(* Logix 5000 project; controller StackLight_Jimmy vendor 1 type 14 code 158 rev 27.11; software revision 27.00 *)

TASK MainTask (continuous, watchdog 500 ms) : MainProgram
TASK SafetyTask (periodic, rate 20 ms, priority 10, watchdog 20 ms, safety) : SafetyProgram

MODULES
   Local : vendor 1 type 14 code 158 (ICP 0, rev 27.11)
      EIP : vendor 1 type 12 code 200 (ICP 2, Ethernet 192.168.1.71, rev 10.1)
         BLCEN_4IOL_2RFID : vendor 48 type 12 code 11502 (Ethernet 192.168.1.30, rev 2.5, StandardDataDriven RPI 20 ms)
      @fcc730f7@:Partner : vendor 1 type 14 code 146 (ICP 1, rev 27.11)
END_MODULES

TYPE Banner_Q4X_Process_Data :   // UDT that records the converted prcoess data.
STRUCT
   Channel_1_Output_State : SINT;   // 0 = Inactive, 1 = Active
   Channel_2_Output_State : SINT;   // 0 = Inactive, 1 = Active
   Sensor_Stability : SINT;   // 0 = No target or Marginal signal, 1 = Stable signal
   Measurement_Value : DINT;   // Distance from sensor face in mm's.
END_STRUCT
END_TYPE

TYPE IO_Link_Port_Data :
STRUCT
   Inputs : SINT[48];
   Outputs : SINT[48];
END_STRUCT
END_TYPE

TYPE UDT_BNI0085_30_22_040 :
STRUCT
   I : UDT_BNI0085_Inputs_30_22_040;
   O : UDT_BNI0085_Outputs_30_22_040;
END_STRUCT
END_TYPE

TYPE UDT_BNI0085_Buzzer_30_22_040 :
STRUCT
   Continuous : BOOL;
   Beep_1Hz : BOOL;   // Beeeeeep---------Beeeeeep---------
   Beep_3Hz : BOOL;   // Beep----Beep----Beep----Beep----
   Short_Beeps_05Hz : BOOL;   // Beep--Beep--Beep--------------------Beep--Beep--Beep----------------
END_STRUCT
END_TYPE

TYPE UDT_BNI0085_Inputs_30_22_040 :
STRUCT
   Error_Code : INT;   // 2=Level Value Out of Range; 4=Num. of Segments Out of Range; 5=Blink Freq. Out of Range; 6=Run Speed Out of Range; 7=Wrong Buzzer Fnction
   Device_OK : BOOL;
   Mismatch_Fault : BOOL;
   Comm_Fault : BOOL;
   Validation_Failed : BOOL;
   Event_1_Error_Code : SINT;
   Event_1_Add_Code_1 : SINT;
   Event_1_Add_Code_2 : SINT;
   Event_2_Error_Code : SINT;
   Event_2_Add_Code_1 : SINT;
   Event_2_Add_Code_2 : SINT;
   Event_3_Error_Code : SINT;
   Event_3_Add_Code_1 : SINT;
   Event_3_Add_Code_2 : SINT;
END_STRUCT
END_TYPE

TYPE UDT_BNI0085_Level_Colors_30_22_040 :
STRUCT
   Green : BOOL;
   Red : BOOL;
   Yellow : BOOL;
   Blue : BOOL;
   Orange : BOOL;
   User_Defined : BOOL;
   White : BOOL;
   Dominant : BOOL;
END_STRUCT
END_TYPE

TYPE UDT_BNI0085_Level_Mode_30_22_040 :
STRUCT
   Enable : BOOL;
   Value : DINT;
   Segment_1 : UDT_BNI0085_Level_Colors_30_22_040;
   Segment_2 : UDT_BNI0085_Level_Colors_30_22_040;
   Segment_3 : UDT_BNI0085_Level_Colors_30_22_040;
   Segment_4 : UDT_BNI0085_Level_Colors_30_22_040;
   Segment_5 : UDT_BNI0085_Level_Colors_30_22_040;
   Fill_Type : BOOL;
END_STRUCT
END_TYPE

TYPE UDT_BNI0085_Outputs_30_22_040 :
STRUCT
   Segment : UDT_BNI0085_Segment_Mode_30_22_040;
   Level : UDT_BNI0085_Level_Mode_30_22_040;
   Runlight : UDT_BNI0085_Runlight_Mode_30_22_040;
   Buzzer : UDT_BNI0085_Buzzer_30_22_040;
END_STRUCT
END_TYPE

TYPE UDT_BNI0085_Runlight_Colors_30_22_040 :
STRUCT
   Green : BOOL;
   Red : BOOL;
   Yellow : BOOL;
   Blue : BOOL;
   Orange : BOOL;
   User_Defined : BOOL;
   White : BOOL;
END_STRUCT
END_TYPE

TYPE UDT_BNI0085_Runlight_Mode_30_22_040 :
STRUCT
   Enable : BOOL;
   Background : UDT_BNI0085_Runlight_Colors_30_22_040;
   Running : UDT_BNI0085_Runlight_Colors_30_22_040;
   Number_of_Segments : SINT;
   Runninng_Speed : SINT;
END_STRUCT
END_TYPE

TYPE UDT_BNI0085_Segment_Colors_30_22_040 :
STRUCT
   Green : BOOL;
   Red : BOOL;
   Yellow : BOOL;
   Blue : BOOL;
   Orange : BOOL;
   User_Defined : BOOL;
   White : BOOL;
   Blink : BOOL;
   Flash : BOOL;
END_STRUCT
END_TYPE

TYPE UDT_BNI0085_Segment_Mode_30_22_040 :
STRUCT
   Enable : BOOL;
   Segment_1 : UDT_BNI0085_Segment_Colors_30_22_040;
   Segment_2 : UDT_BNI0085_Segment_Colors_30_22_040;
   Segment_3 : UDT_BNI0085_Segment_Colors_30_22_040;
   Segment_4 : UDT_BNI0085_Segment_Colors_30_22_040;
   Segment_5 : UDT_BNI0085_Segment_Colors_30_22_040;
   Number_of_Segments : SINT;
   Blink_Frequency : SINT;
END_STRUCT
END_TYPE

ADD_ON_INSTRUCTION AOI_BNI0085_30_22_040   (* revision 0.4 *)
VAR_IN_OUT
   IO_Link_Port_Data : IO_Link_Port_Data; {required}
   BNI0085_Mapped_Data : UDT_BNI0085_30_22_040; {required}
END_VAR
VAR
   Segment_Array : SINT[8]; {access None}
   Level_Array : SINT[8]; {access None}
   Runlight_Array : SINT[8]; {access None}
END_VAR

ROUTINE Logic   (* ladder *)
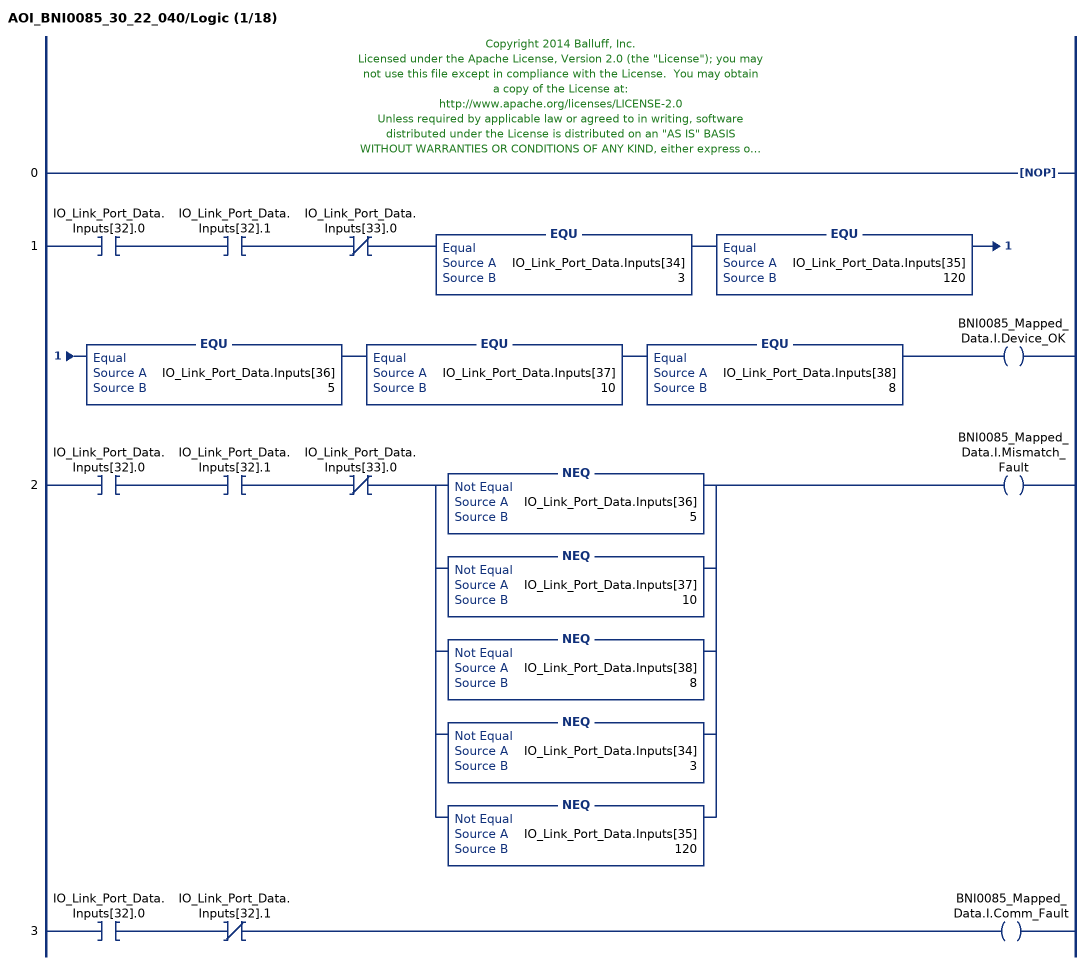
   // Copyright 2014 Balluff, Inc.
   // Licensed under the Apache License, Version 2.0 (the "License"); you may
   // not use this file except in compliance with the License.  You may obtain
   // a copy of the License at:
   // http://www.apache.org/licenses/LICENSE-2.0
   // Unless required by applicable law or agreed to in writing, software
   // distributed under the License is distributed on an "AS IS" BASIS
   // WITHOUT WARRANTIES OR CONDITIONS OF ANY KIND, either express or
   // implied.  See the License for the specific language governing
   // permissions and limitations under the License.
   0: NOP();
   1: XIC(IO_Link_Port_Data.Inputs[32].0)XIC(IO_Link_Port_Data.Inputs[32].1)XIO(IO_Link_Port_Data.Inputs[33].0)EQU(IO_Link_Port_Data.Inputs[34],3)EQU(IO_Link_Port_Data.Inputs[35],120)EQU(IO_Link_Port_Data.Inputs[36],5)EQU(IO_Link_Port_Data.Inputs[37],10)EQU(IO_Link_Port_Data.Inputs[38],8)OTE(BNI0085_Mapped_Data.I.Device_OK);
   2: XIC(IO_Link_Port_Data.Inputs[32].0)XIC(IO_Link_Port_Data.Inputs[32].1)XIO(IO_Link_Port_Data.Inputs[33].0)[NEQ(IO_Link_Port_Data.Inputs[36],5) ,NEQ(IO_Link_Port_Data.Inputs[37],10) ,NEQ(IO_Link_Port_Data.Inputs[38],8) ,NEQ(IO_Link_Port_Data.Inputs[34],3) ,NEQ(IO_Link_Port_Data.Inputs[35],120) ]OTE(BNI0085_Mapped_Data.I.Mismatch_Fault);
   3: XIC(IO_Link_Port_Data.Inputs[32].0)XIO(IO_Link_Port_Data.Inputs[32].1)OTE(BNI0085_Mapped_Data.I.Comm_Fault);
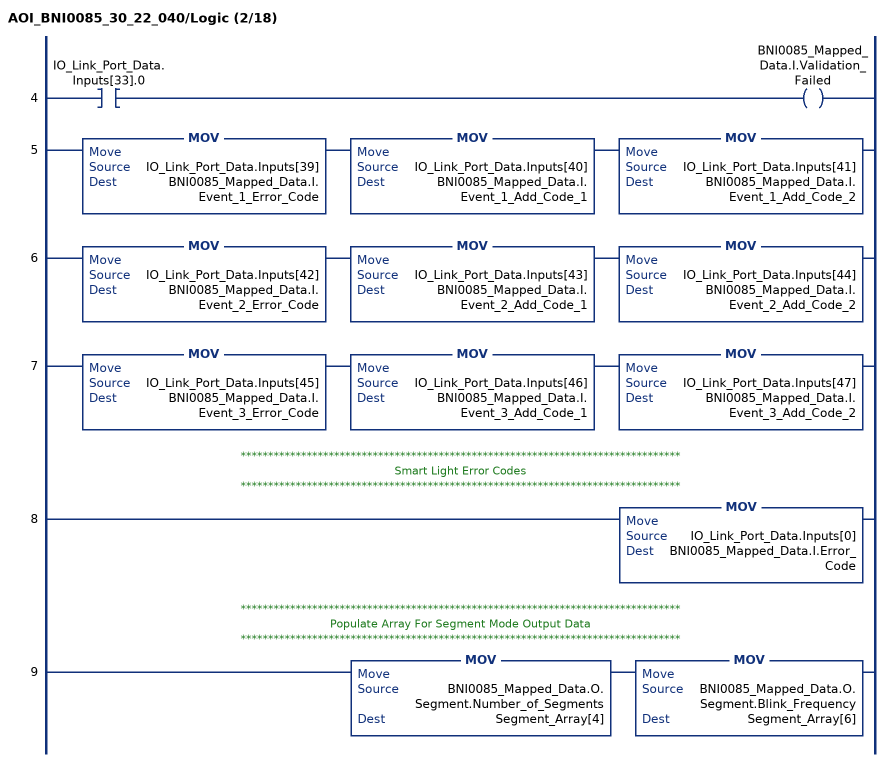
   4: XIC(IO_Link_Port_Data.Inputs[33].0)OTE(BNI0085_Mapped_Data.I.Validation_Failed);
   5: MOV(IO_Link_Port_Data.Inputs[39],BNI0085_Mapped_Data.I.Event_1_Error_Code)MOV(IO_Link_Port_Data.Inputs[40],BNI0085_Mapped_Data.I.Event_1_Add_Code_1)MOV(IO_Link_Port_Data.Inputs[41],BNI0085_Mapped_Data.I.Event_1_Add_Code_2);
   6: MOV(IO_Link_Port_Data.Inputs[42],BNI0085_Mapped_Data.I.Event_2_Error_Code)MOV(IO_Link_Port_Data.Inputs[43],BNI0085_Mapped_Data.I.Event_2_Add_Code_1)MOV(IO_Link_Port_Data.Inputs[44],BNI0085_Mapped_Data.I.Event_2_Add_Code_2);
   7: MOV(IO_Link_Port_Data.Inputs[45],BNI0085_Mapped_Data.I.Event_3_Error_Code)MOV(IO_Link_Port_Data.Inputs[46],BNI0085_Mapped_Data.I.Event_3_Add_Code_1)MOV(IO_Link_Port_Data.Inputs[47],BNI0085_Mapped_Data.I.Event_3_Add_Code_2);
   // ********************************************************************************
   // Smart Light Error Codes
   // ********************************************************************************
   8: MOV(IO_Link_Port_Data.Inputs[0],BNI0085_Mapped_Data.I.Error_Code);
   // ********************************************************************************
   // Populate Array For Segment Mode Output Data
   // ********************************************************************************
   9: MOV(BNI0085_Mapped_Data.O.Segment.Number_of_Segments,Segment_Array[4])MOV(BNI0085_Mapped_Data.O.Segment.Blink_Frequency,Segment_Array[6]);
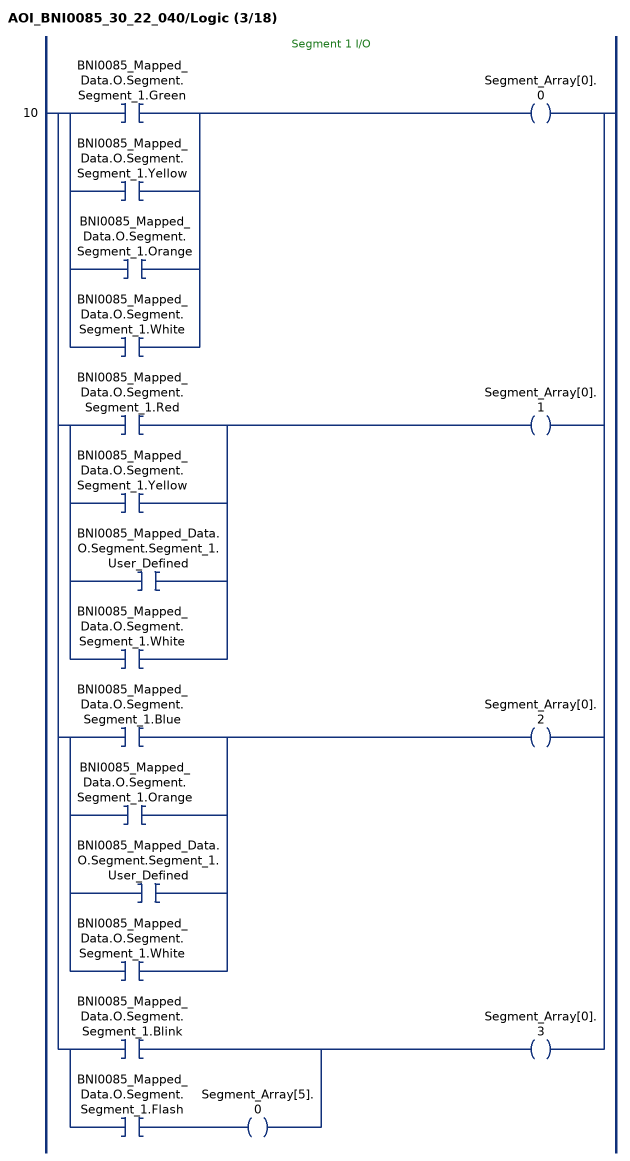
   // Segment 1 I/O
   10: [[XIC(BNI0085_Mapped_Data.O.Segment.Segment_1.Green) ,XIC(BNI0085_Mapped_Data.O.Segment.Segment_1.Yellow) ,XIC(BNI0085_Mapped_Data.O.Segment.Segment_1.Orange) ,XIC(BNI0085_Mapped_Data.O.Segment.Segment_1.White) ] OTE(Segment_Array[0].0) ,[XIC(BNI0085_Mapped_Data.O.Segment.Segment_1.Red) ,XIC(BNI0085_Mapped_Data.O.Segment.Segment_1.Yellow) ,XIC(BNI0085_Mapped_Data.O.Segment.Segment_1.User_Defined) ,XIC(BNI0085_Mapped_Data.O.Segment.Segment_1.White) ] OTE(Segment_Array[0].1) ,[XIC(BNI0085_Mapped_Data.O.Segment.Segment_1.Blue) ,XIC(BNI0085_Mapped_Data.O.Segment.Segment_1.Orange) ,XIC(BNI0085_Mapped_Data.O.Segment.Segment_1.User_Defined) ,XIC(BNI0085_Mapped_Data.O.Segment.Segment_1.White) ] OTE(Segment_Array[0].2) ,[XIC(BNI0085_Mapped_Data.O.Segment.Segment_1.Blink) ,XIC(BNI0085_Mapped_Data.O.Segment.Segment_1.Flash) OTE(Segment_Array[5].0) ] OTE(Segment_Array[0].3) ];
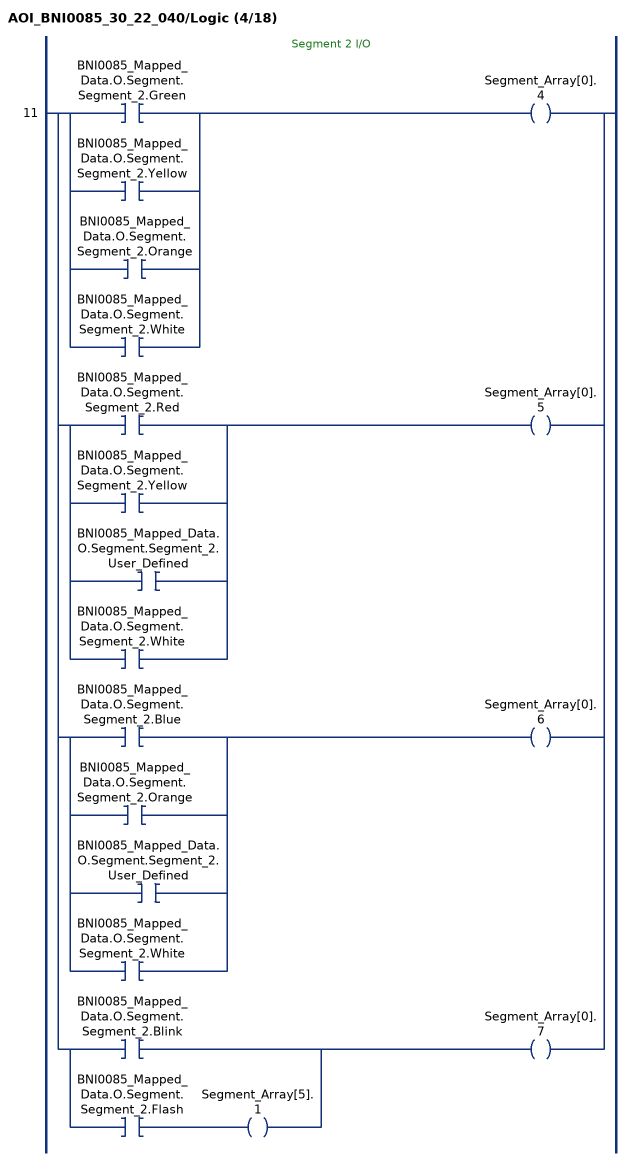
   // Segment 2 I/O
   11: [[XIC(BNI0085_Mapped_Data.O.Segment.Segment_2.Green) ,XIC(BNI0085_Mapped_Data.O.Segment.Segment_2.Yellow) ,XIC(BNI0085_Mapped_Data.O.Segment.Segment_2.Orange) ,XIC(BNI0085_Mapped_Data.O.Segment.Segment_2.White) ] OTE(Segment_Array[0].4) ,[XIC(BNI0085_Mapped_Data.O.Segment.Segment_2.Red) ,XIC(BNI0085_Mapped_Data.O.Segment.Segment_2.Yellow) ,XIC(BNI0085_Mapped_Data.O.Segment.Segment_2.User_Defined) ,XIC(BNI0085_Mapped_Data.O.Segment.Segment_2.White) ] OTE(Segment_Array[0].5) ,[XIC(BNI0085_Mapped_Data.O.Segment.Segment_2.Blue) ,XIC(BNI0085_Mapped_Data.O.Segment.Segment_2.Orange) ,XIC(BNI0085_Mapped_Data.O.Segment.Segment_2.User_Defined) ,XIC(BNI0085_Mapped_Data.O.Segment.Segment_2.White) ] OTE(Segment_Array[0].6) ,[XIC(BNI0085_Mapped_Data.O.Segment.Segment_2.Blink) ,XIC(BNI0085_Mapped_Data.O.Segment.Segment_2.Flash) OTE(Segment_Array[5].1) ] OTE(Segment_Array[0].7) ];
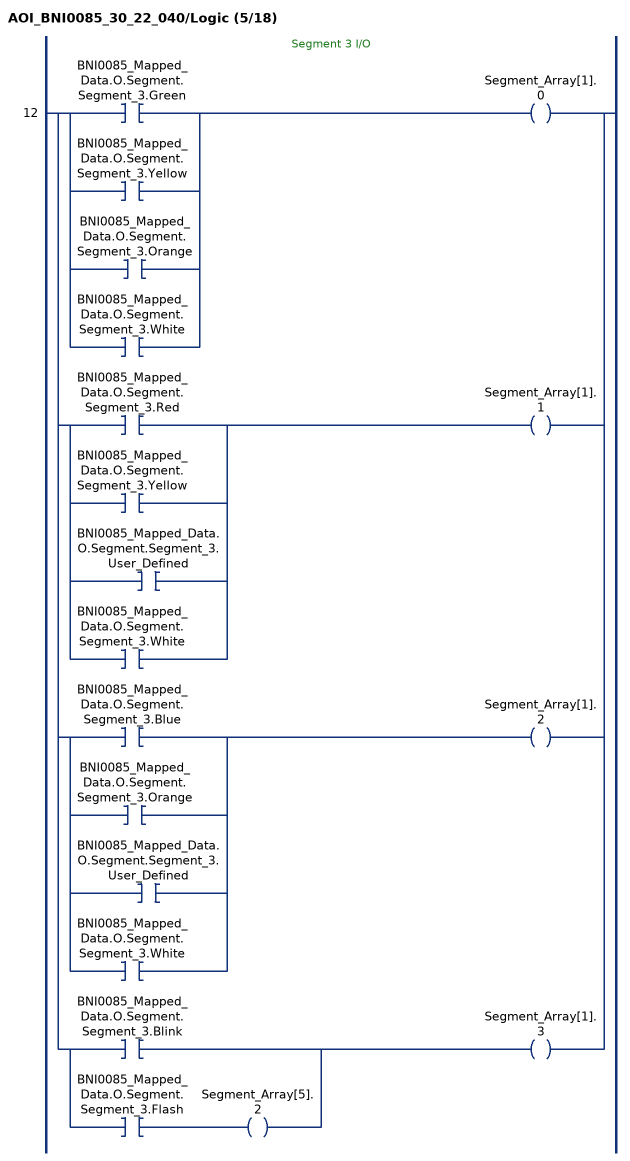
   // Segment 3 I/O
   12: [[XIC(BNI0085_Mapped_Data.O.Segment.Segment_3.Green) ,XIC(BNI0085_Mapped_Data.O.Segment.Segment_3.Yellow) ,XIC(BNI0085_Mapped_Data.O.Segment.Segment_3.Orange) ,XIC(BNI0085_Mapped_Data.O.Segment.Segment_3.White) ] OTE(Segment_Array[1].0) ,[XIC(BNI0085_Mapped_Data.O.Segment.Segment_3.Red) ,XIC(BNI0085_Mapped_Data.O.Segment.Segment_3.Yellow) ,XIC(BNI0085_Mapped_Data.O.Segment.Segment_3.User_Defined) ,XIC(BNI0085_Mapped_Data.O.Segment.Segment_3.White) ] OTE(Segment_Array[1].1) ,[XIC(BNI0085_Mapped_Data.O.Segment.Segment_3.Blue) ,XIC(BNI0085_Mapped_Data.O.Segment.Segment_3.Orange) ,XIC(BNI0085_Mapped_Data.O.Segment.Segment_3.User_Defined) ,XIC(BNI0085_Mapped_Data.O.Segment.Segment_3.White) ] OTE(Segment_Array[1].2) ,[XIC(BNI0085_Mapped_Data.O.Segment.Segment_3.Blink) ,XIC(BNI0085_Mapped_Data.O.Segment.Segment_3.Flash) OTE(Segment_Array[5].2) ] OTE(Segment_Array[1].3) ];
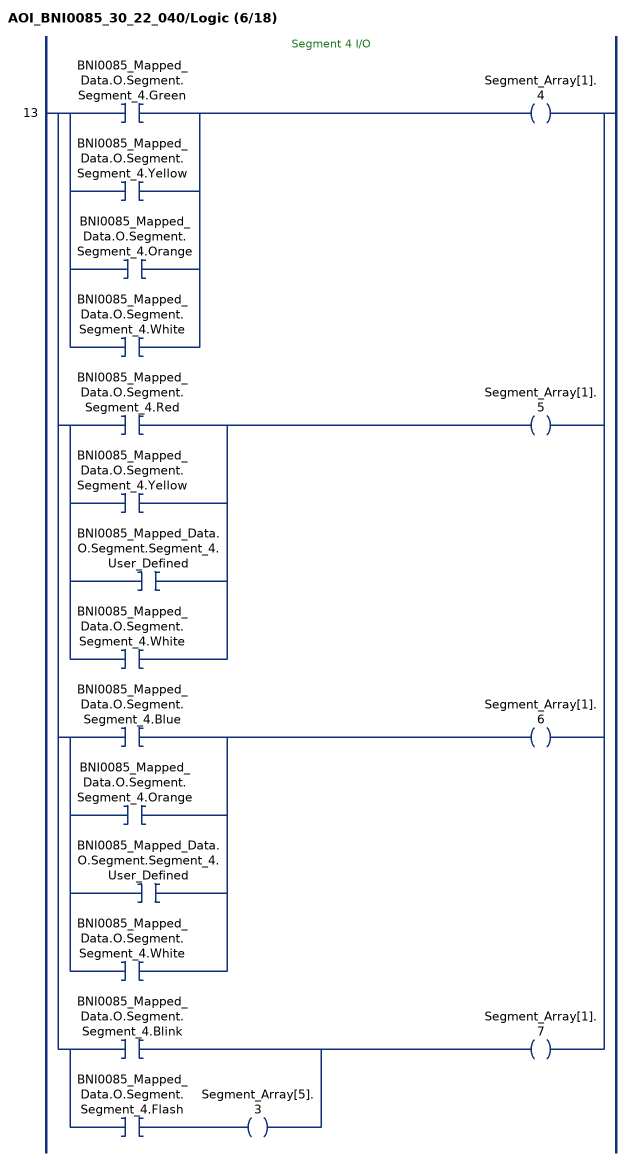
   // Segment 4 I/O
   13: [[XIC(BNI0085_Mapped_Data.O.Segment.Segment_4.Green) ,XIC(BNI0085_Mapped_Data.O.Segment.Segment_4.Yellow) ,XIC(BNI0085_Mapped_Data.O.Segment.Segment_4.Orange) ,XIC(BNI0085_Mapped_Data.O.Segment.Segment_4.White) ] OTE(Segment_Array[1].4) ,[XIC(BNI0085_Mapped_Data.O.Segment.Segment_4.Red) ,XIC(BNI0085_Mapped_Data.O.Segment.Segment_4.Yellow) ,XIC(BNI0085_Mapped_Data.O.Segment.Segment_4.User_Defined) ,XIC(BNI0085_Mapped_Data.O.Segment.Segment_4.White) ] OTE(Segment_Array[1].5) ,[XIC(BNI0085_Mapped_Data.O.Segment.Segment_4.Blue) ,XIC(BNI0085_Mapped_Data.O.Segment.Segment_4.Orange) ,XIC(BNI0085_Mapped_Data.O.Segment.Segment_4.User_Defined) ,XIC(BNI0085_Mapped_Data.O.Segment.Segment_4.White) ] OTE(Segment_Array[1].6) ,[XIC(BNI0085_Mapped_Data.O.Segment.Segment_4.Blink) ,XIC(BNI0085_Mapped_Data.O.Segment.Segment_4.Flash) OTE(Segment_Array[5].3) ] OTE(Segment_Array[1].7) ];
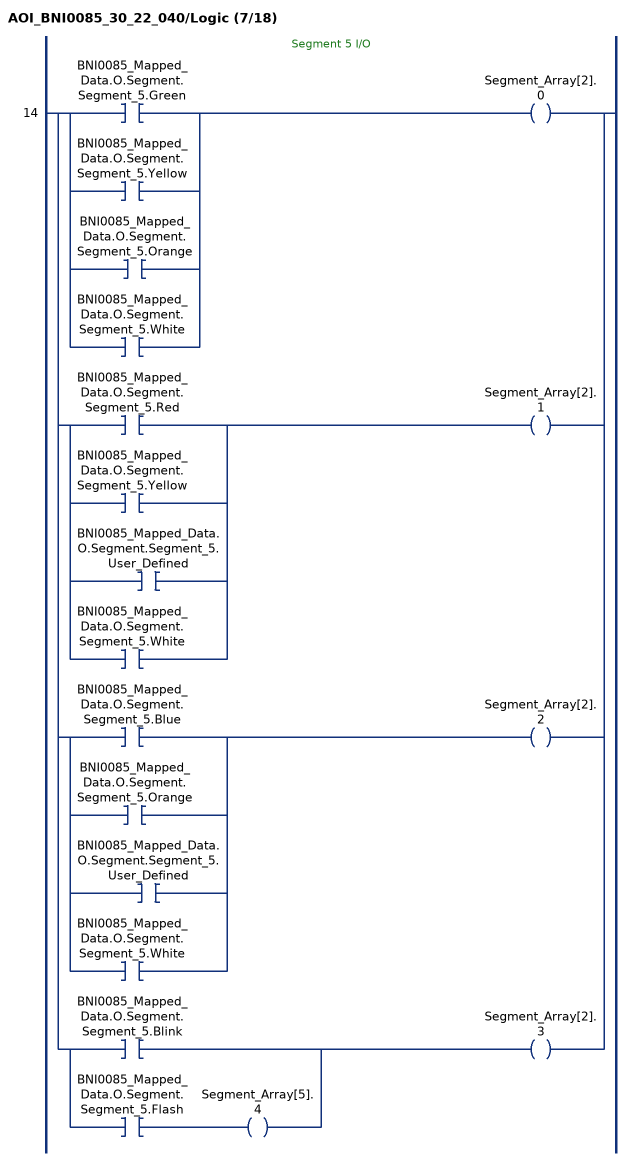
   // Segment 5 I/O
   14: [[XIC(BNI0085_Mapped_Data.O.Segment.Segment_5.Green) ,XIC(BNI0085_Mapped_Data.O.Segment.Segment_5.Yellow) ,XIC(BNI0085_Mapped_Data.O.Segment.Segment_5.Orange) ,XIC(BNI0085_Mapped_Data.O.Segment.Segment_5.White) ] OTE(Segment_Array[2].0) ,[XIC(BNI0085_Mapped_Data.O.Segment.Segment_5.Red) ,XIC(BNI0085_Mapped_Data.O.Segment.Segment_5.Yellow) ,XIC(BNI0085_Mapped_Data.O.Segment.Segment_5.User_Defined) ,XIC(BNI0085_Mapped_Data.O.Segment.Segment_5.White) ] OTE(Segment_Array[2].1) ,[XIC(BNI0085_Mapped_Data.O.Segment.Segment_5.Blue) ,XIC(BNI0085_Mapped_Data.O.Segment.Segment_5.Orange) ,XIC(BNI0085_Mapped_Data.O.Segment.Segment_5.User_Defined) ,XIC(BNI0085_Mapped_Data.O.Segment.Segment_5.White) ] OTE(Segment_Array[2].2) ,[XIC(BNI0085_Mapped_Data.O.Segment.Segment_5.Blink) ,XIC(BNI0085_Mapped_Data.O.Segment.Segment_5.Flash) OTE(Segment_Array[5].4) ] OTE(Segment_Array[2].3) ];
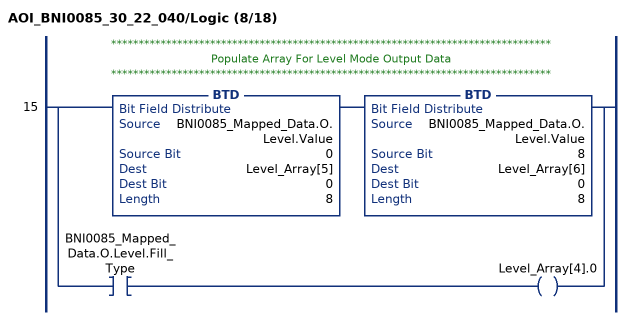
   // ********************************************************************************
   // Populate Array For Level Mode Output Data
   // ********************************************************************************
   15: [BTD(BNI0085_Mapped_Data.O.Level.Value,0,Level_Array[5],0,8) BTD(BNI0085_Mapped_Data.O.Level.Value,8,Level_Array[6],0,8) ,XIC(BNI0085_Mapped_Data.O.Level.Fill_Type) OTE(Level_Array[4].0) ];
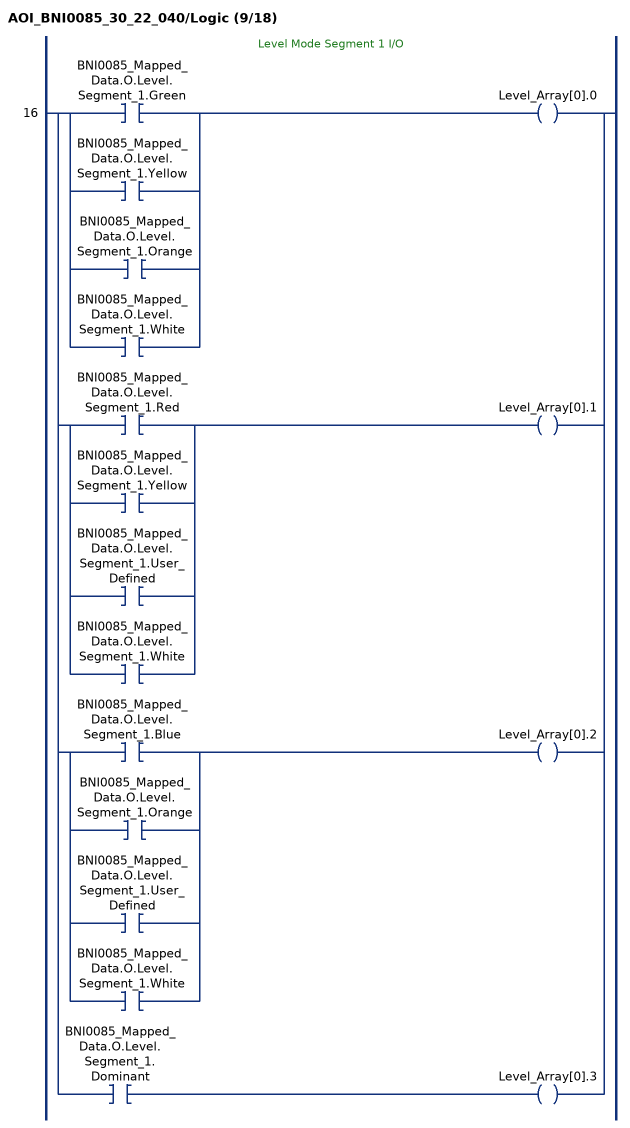
   // Level Mode Segment 1 I/O
   16: [[XIC(BNI0085_Mapped_Data.O.Level.Segment_1.Green) ,XIC(BNI0085_Mapped_Data.O.Level.Segment_1.Yellow) ,XIC(BNI0085_Mapped_Data.O.Level.Segment_1.Orange) ,XIC(BNI0085_Mapped_Data.O.Level.Segment_1.White) ] OTE(Level_Array[0].0) ,[XIC(BNI0085_Mapped_Data.O.Level.Segment_1.Red) ,XIC(BNI0085_Mapped_Data.O.Level.Segment_1.Yellow) ,XIC(BNI0085_Mapped_Data.O.Level.Segment_1.User_Defined) ,XIC(BNI0085_Mapped_Data.O.Level.Segment_1.White) ] OTE(Level_Array[0].1) ,[XIC(BNI0085_Mapped_Data.O.Level.Segment_1.Blue) ,XIC(BNI0085_Mapped_Data.O.Level.Segment_1.Orange) ,XIC(BNI0085_Mapped_Data.O.Level.Segment_1.User_Defined) ,XIC(BNI0085_Mapped_Data.O.Level.Segment_1.White) ] OTE(Level_Array[0].2) ,XIC(BNI0085_Mapped_Data.O.Level.Segment_1.Dominant) OTE(Level_Array[0].3) ];
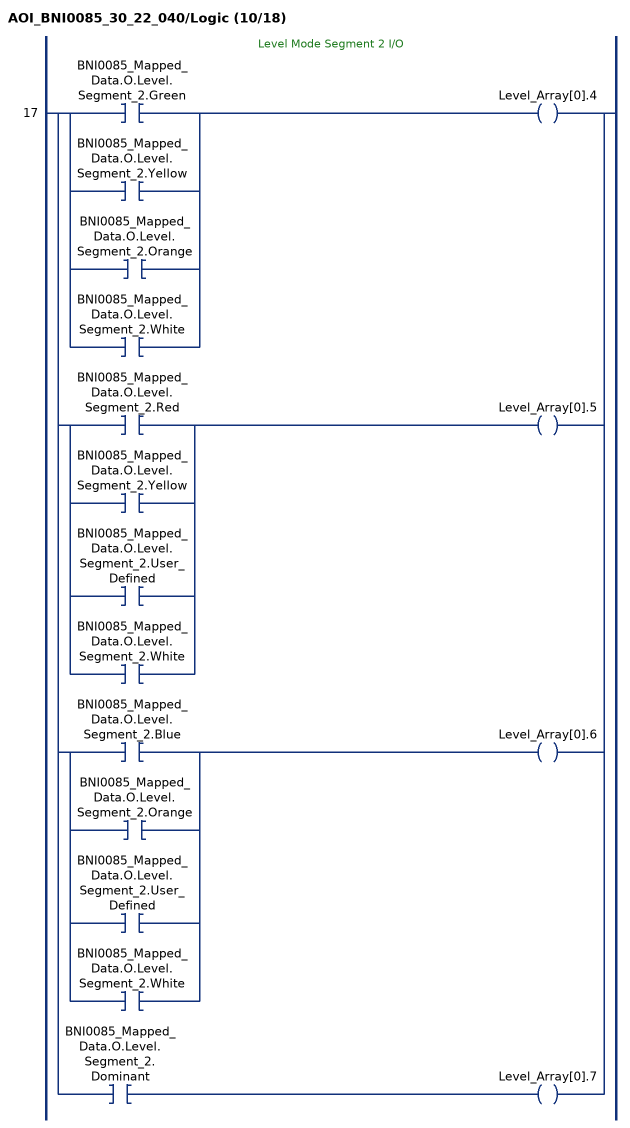
   // Level Mode Segment 2 I/O
   17: [[XIC(BNI0085_Mapped_Data.O.Level.Segment_2.Green) ,XIC(BNI0085_Mapped_Data.O.Level.Segment_2.Yellow) ,XIC(BNI0085_Mapped_Data.O.Level.Segment_2.Orange) ,XIC(BNI0085_Mapped_Data.O.Level.Segment_2.White) ] OTE(Level_Array[0].4) ,[XIC(BNI0085_Mapped_Data.O.Level.Segment_2.Red) ,XIC(BNI0085_Mapped_Data.O.Level.Segment_2.Yellow) ,XIC(BNI0085_Mapped_Data.O.Level.Segment_2.User_Defined) ,XIC(BNI0085_Mapped_Data.O.Level.Segment_2.White) ] OTE(Level_Array[0].5) ,[XIC(BNI0085_Mapped_Data.O.Level.Segment_2.Blue) ,XIC(BNI0085_Mapped_Data.O.Level.Segment_2.Orange) ,XIC(BNI0085_Mapped_Data.O.Level.Segment_2.User_Defined) ,XIC(BNI0085_Mapped_Data.O.Level.Segment_2.White) ] OTE(Level_Array[0].6) ,XIC(BNI0085_Mapped_Data.O.Level.Segment_2.Dominant) OTE(Level_Array[0].7) ];
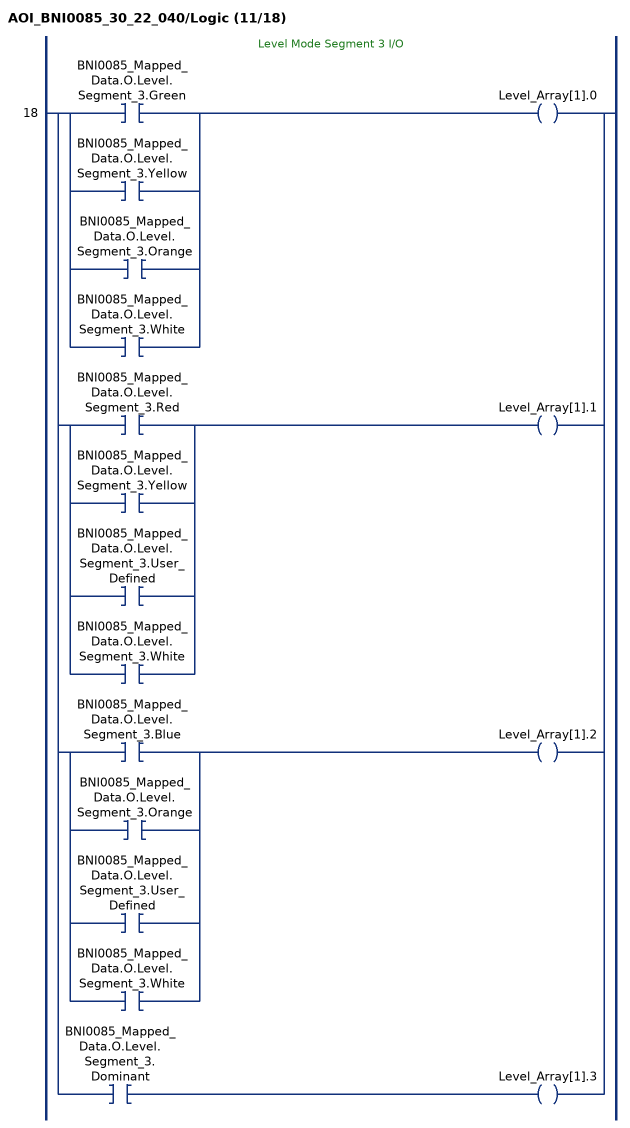
   // Level Mode Segment 3 I/O
   18: [[XIC(BNI0085_Mapped_Data.O.Level.Segment_3.Green) ,XIC(BNI0085_Mapped_Data.O.Level.Segment_3.Yellow) ,XIC(BNI0085_Mapped_Data.O.Level.Segment_3.Orange) ,XIC(BNI0085_Mapped_Data.O.Level.Segment_3.White) ] OTE(Level_Array[1].0) ,[XIC(BNI0085_Mapped_Data.O.Level.Segment_3.Red) ,XIC(BNI0085_Mapped_Data.O.Level.Segment_3.Yellow) ,XIC(BNI0085_Mapped_Data.O.Level.Segment_3.User_Defined) ,XIC(BNI0085_Mapped_Data.O.Level.Segment_3.White) ] OTE(Level_Array[1].1) ,[XIC(BNI0085_Mapped_Data.O.Level.Segment_3.Blue) ,XIC(BNI0085_Mapped_Data.O.Level.Segment_3.Orange) ,XIC(BNI0085_Mapped_Data.O.Level.Segment_3.User_Defined) ,XIC(BNI0085_Mapped_Data.O.Level.Segment_3.White) ] OTE(Level_Array[1].2) ,XIC(BNI0085_Mapped_Data.O.Level.Segment_3.Dominant) OTE(Level_Array[1].3) ];
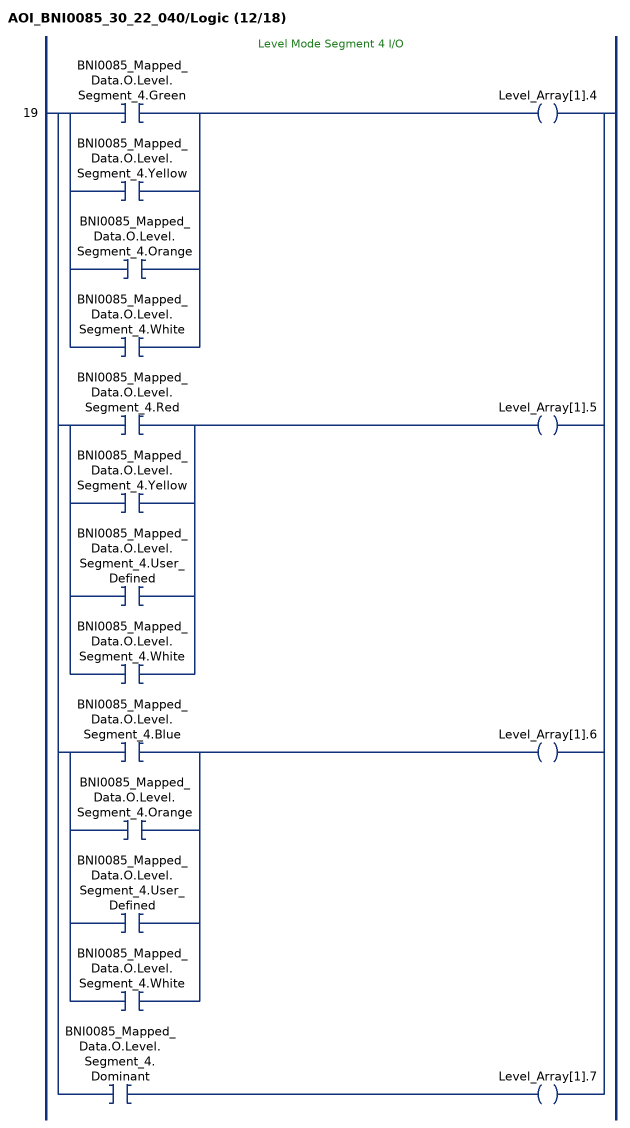
   // Level Mode Segment 4 I/O
   19: [[XIC(BNI0085_Mapped_Data.O.Level.Segment_4.Green) ,XIC(BNI0085_Mapped_Data.O.Level.Segment_4.Yellow) ,XIC(BNI0085_Mapped_Data.O.Level.Segment_4.Orange) ,XIC(BNI0085_Mapped_Data.O.Level.Segment_4.White) ] OTE(Level_Array[1].4) ,[XIC(BNI0085_Mapped_Data.O.Level.Segment_4.Red) ,XIC(BNI0085_Mapped_Data.O.Level.Segment_4.Yellow) ,XIC(BNI0085_Mapped_Data.O.Level.Segment_4.User_Defined) ,XIC(BNI0085_Mapped_Data.O.Level.Segment_4.White) ] OTE(Level_Array[1].5) ,[XIC(BNI0085_Mapped_Data.O.Level.Segment_4.Blue) ,XIC(BNI0085_Mapped_Data.O.Level.Segment_4.Orange) ,XIC(BNI0085_Mapped_Data.O.Level.Segment_4.User_Defined) ,XIC(BNI0085_Mapped_Data.O.Level.Segment_4.White) ] OTE(Level_Array[1].6) ,XIC(BNI0085_Mapped_Data.O.Level.Segment_4.Dominant) OTE(Level_Array[1].7) ];
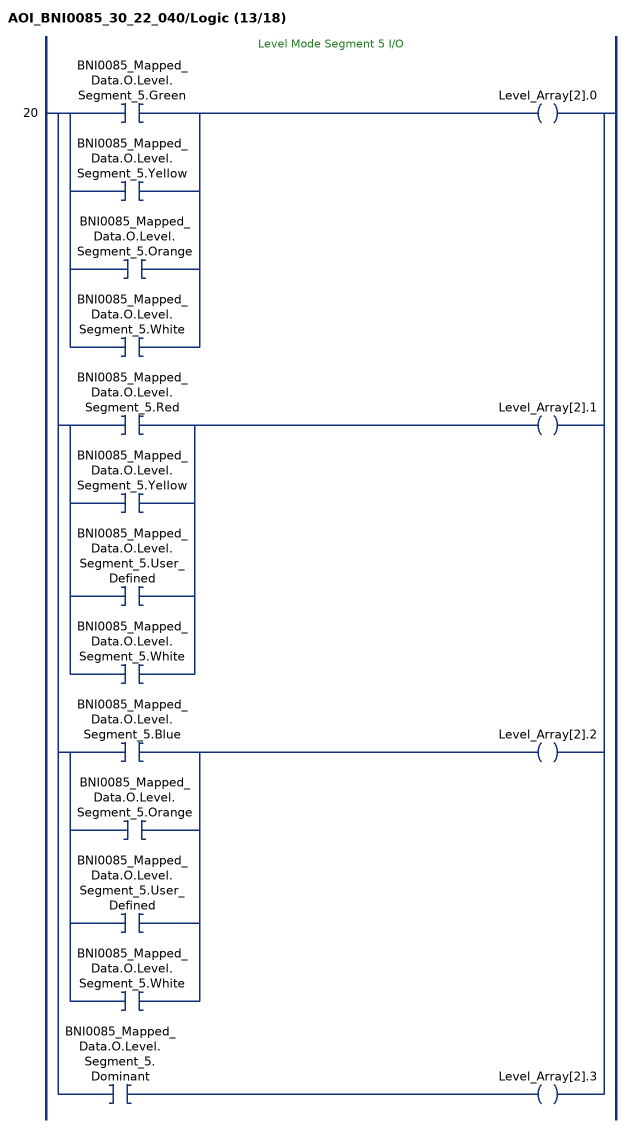
   // Level Mode Segment 5 I/O
   20: [[XIC(BNI0085_Mapped_Data.O.Level.Segment_5.Green) ,XIC(BNI0085_Mapped_Data.O.Level.Segment_5.Yellow) ,XIC(BNI0085_Mapped_Data.O.Level.Segment_5.Orange) ,XIC(BNI0085_Mapped_Data.O.Level.Segment_5.White) ] OTE(Level_Array[2].0) ,[XIC(BNI0085_Mapped_Data.O.Level.Segment_5.Red) ,XIC(BNI0085_Mapped_Data.O.Level.Segment_5.Yellow) ,XIC(BNI0085_Mapped_Data.O.Level.Segment_5.User_Defined) ,XIC(BNI0085_Mapped_Data.O.Level.Segment_5.White) ] OTE(Level_Array[2].1) ,[XIC(BNI0085_Mapped_Data.O.Level.Segment_5.Blue) ,XIC(BNI0085_Mapped_Data.O.Level.Segment_5.Orange) ,XIC(BNI0085_Mapped_Data.O.Level.Segment_5.User_Defined) ,XIC(BNI0085_Mapped_Data.O.Level.Segment_5.White) ] OTE(Level_Array[2].2) ,XIC(BNI0085_Mapped_Data.O.Level.Segment_5.Dominant) OTE(Level_Array[2].3) ];
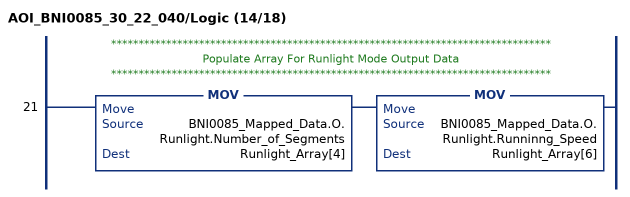
   // ********************************************************************************
   // Populate Array For Runlight Mode Output Data
   // ********************************************************************************
   21: MOV(BNI0085_Mapped_Data.O.Runlight.Number_of_Segments,Runlight_Array[4])MOV(BNI0085_Mapped_Data.O.Runlight.Runninng_Speed,Runlight_Array[6]);
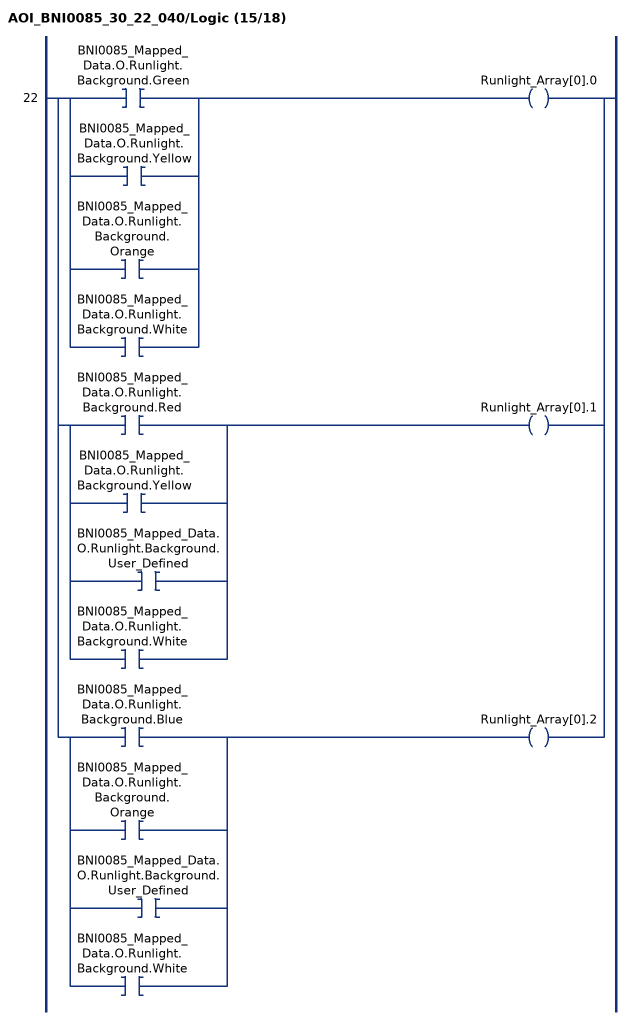
   22: [[XIC(BNI0085_Mapped_Data.O.Runlight.Background.Green) ,XIC(BNI0085_Mapped_Data.O.Runlight.Background.Yellow) ,XIC(BNI0085_Mapped_Data.O.Runlight.Background.Orange) ,XIC(BNI0085_Mapped_Data.O.Runlight.Background.White) ] OTE(Runlight_Array[0].0) ,[XIC(BNI0085_Mapped_Data.O.Runlight.Background.Red) ,XIC(BNI0085_Mapped_Data.O.Runlight.Background.Yellow) ,XIC(BNI0085_Mapped_Data.O.Runlight.Background.User_Defined) ,XIC(BNI0085_Mapped_Data.O.Runlight.Background.White) ] OTE(Runlight_Array[0].1) ,[XIC(BNI0085_Mapped_Data.O.Runlight.Background.Blue) ,XIC(BNI0085_Mapped_Data.O.Runlight.Background.Orange) ,XIC(BNI0085_Mapped_Data.O.Runlight.Background.User_Defined) ,XIC(BNI0085_Mapped_Data.O.Runlight.Background.White) ] OTE(Runlight_Array[0].2) ];
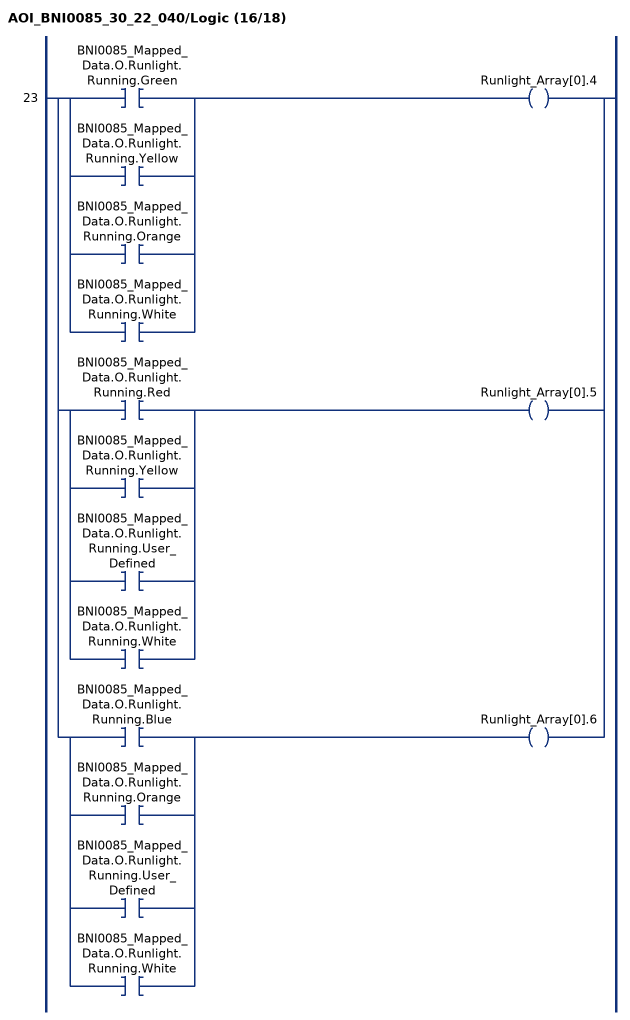
   23: [[XIC(BNI0085_Mapped_Data.O.Runlight.Running.Green) ,XIC(BNI0085_Mapped_Data.O.Runlight.Running.Yellow) ,XIC(BNI0085_Mapped_Data.O.Runlight.Running.Orange) ,XIC(BNI0085_Mapped_Data.O.Runlight.Running.White) ] OTE(Runlight_Array[0].4) ,[XIC(BNI0085_Mapped_Data.O.Runlight.Running.Red) ,XIC(BNI0085_Mapped_Data.O.Runlight.Running.Yellow) ,XIC(BNI0085_Mapped_Data.O.Runlight.Running.User_Defined) ,XIC(BNI0085_Mapped_Data.O.Runlight.Running.White) ] OTE(Runlight_Array[0].5) ,[XIC(BNI0085_Mapped_Data.O.Runlight.Running.Blue) ,XIC(BNI0085_Mapped_Data.O.Runlight.Running.Orange) ,XIC(BNI0085_Mapped_Data.O.Runlight.Running.User_Defined) ,XIC(BNI0085_Mapped_Data.O.Runlight.Running.White) ] OTE(Runlight_Array[0].6) ];
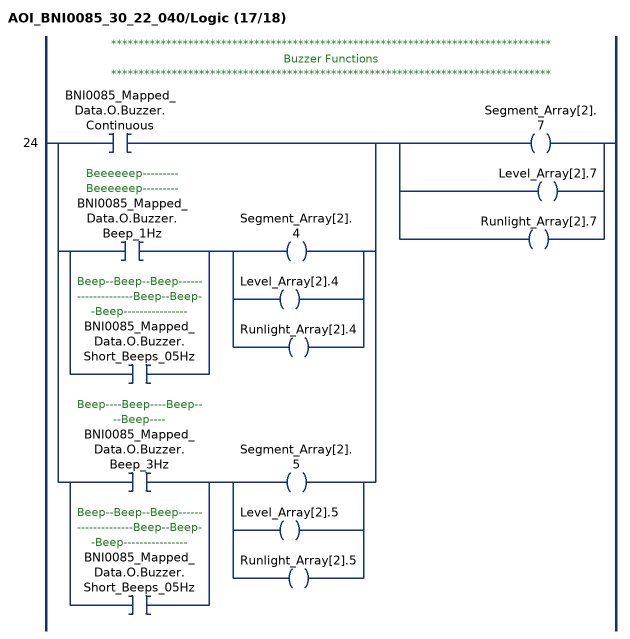
   // ********************************************************************************
   // Buzzer Functions
   // ********************************************************************************
   24: [XIC(BNI0085_Mapped_Data.O.Buzzer.Continuous) ,[XIC(BNI0085_Mapped_Data.O.Buzzer.Beep_1Hz) ,XIC(BNI0085_Mapped_Data.O.Buzzer.Short_Beeps_05Hz) ] [OTE(Segment_Array[2].4) ,OTE(Level_Array[2].4) ,OTE(Runlight_Array[2].4) ] ,[XIC(BNI0085_Mapped_Data.O.Buzzer.Beep_3Hz) ,XIC(BNI0085_Mapped_Data.O.Buzzer.Short_Beeps_05Hz) ] [OTE(Segment_Array[2].5) ,OTE(Level_Array[2].5) ,OTE(Runlight_Array[2].5) ] ][OTE(Segment_Array[2].7) ,OTE(Level_Array[2].7) ,OTE(Runlight_Array[2].7) ];
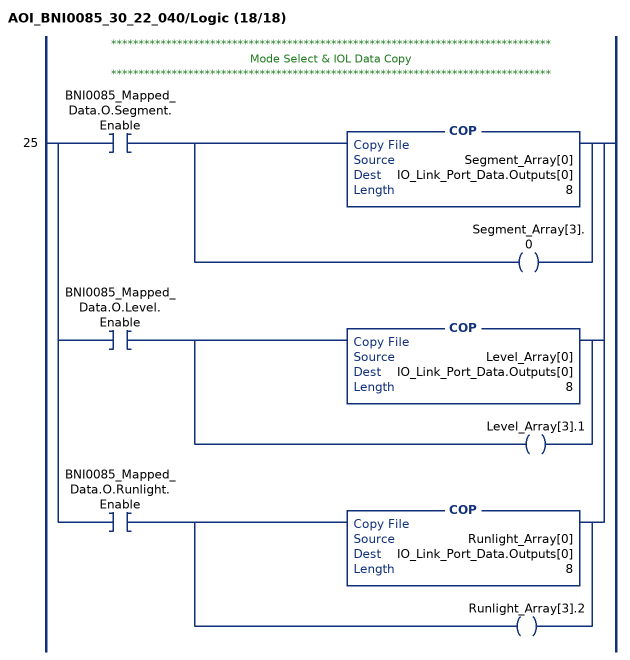
   // ********************************************************************************
   // Mode Select & IOL Data Copy
   // ********************************************************************************
   25: [XIC(BNI0085_Mapped_Data.O.Segment.Enable) [COP(Segment_Array[0],IO_Link_Port_Data.Outputs[0],8) ,OTE(Segment_Array[3].0) ] ,XIC(BNI0085_Mapped_Data.O.Level.Enable) [COP(Level_Array[0],IO_Link_Port_Data.Outputs[0],8) ,OTE(Level_Array[3].1) ] ,XIC(BNI0085_Mapped_Data.O.Runlight.Enable) [COP(Runlight_Array[0],IO_Link_Port_Data.Outputs[0],8) ,OTE(Runlight_Array[3].2) ] ];
END_ROUTINE
END_ADD_ON_INSTRUCTION

ADD_ON_INSTRUCTION Banner_Q4X_Process_Data_AOI_BC   (* revision 1.0, vendor Banner Engineering *)
// Takes the raw SINT information and converts that data into actual information.
VAR_IN_OUT
   SINT0 : SINT; {required}
   SINT1 : SINT; {required}
   PROCESS_DATA : Banner_Q4X_Process_Data; {required}
END_VAR
VAR
   Temp_Measurement : DINT; {access None}
END_VAR

ROUTINE Logic   (* ladder *)
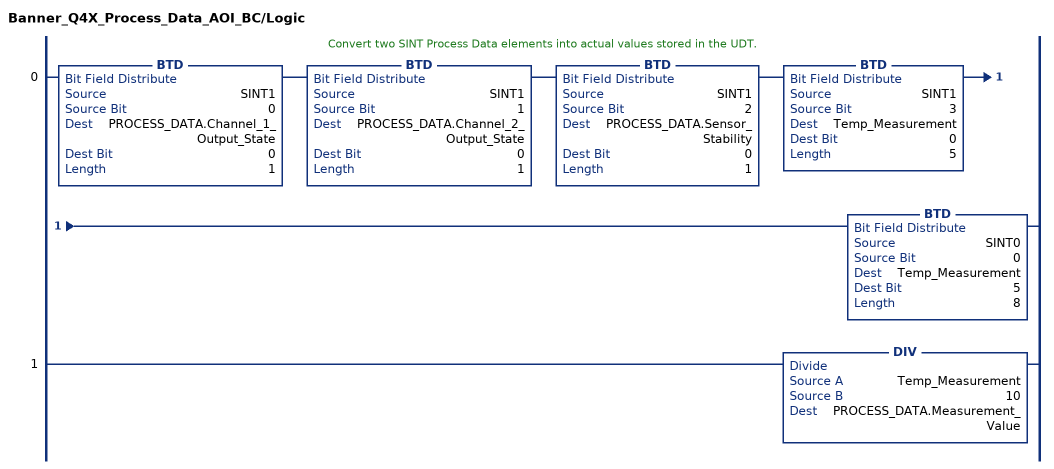
   // Convert two SINT Process Data elements into actual values stored in the UDT.
   0: BTD(SINT1,0,PROCESS_DATA.Channel_1_Output_State,0,1)BTD(SINT1,1,PROCESS_DATA.Channel_2_Output_State,0,1)BTD(SINT1,2,PROCESS_DATA.Sensor_Stability,0,1)BTD(SINT1,3,Temp_Measurement,0,5)BTD(SINT0,0,Temp_Measurement,5,8);
   1: DIV(Temp_Measurement,10,PROCESS_DATA.Measurement_Value);
END_ROUTINE
END_ADD_ON_INSTRUCTION

VAR_GLOBAL   (* controller tags *)
   Adjusted_Value : DINT;
   Banner_input_0 : SINT;
   Banner_input_1 : SINT;
   Banner_Q4x_data : Banner_Q4X_Process_Data_AOI_BC;
   Banner_Q4x_mapped : Banner_Q4X_Process_Data;
   IOL_Port_Data : IO_Link_Port_Data := (Inputs[32] := 3, Inputs[34] := 3, Inputs[35] := 120, Inputs[36] := 5, Inputs[37] := 10, Inputs[38] := 8, Outputs[0] := 4, Outputs[3] := 1, Outputs[4] := 36);
   Low_mask : INT := 255;
   Stack_Light_AOI : AOI_BNI0085_30_22_040;
   Stack_Light_Mapped_Data : UDT_BNI0085_30_22_040 := (I.Device_OK := 1, O.Segment.Enable := 1, O.Segment.Segment_1.Blue := 1, O.Segment.Number_of_Segments := 36);
   temp_swap : INT;
END_VAR

PROGRAM MainProgram   (* main routine MainRoutine *)

ROUTINE MainRoutine   (* ladder *)
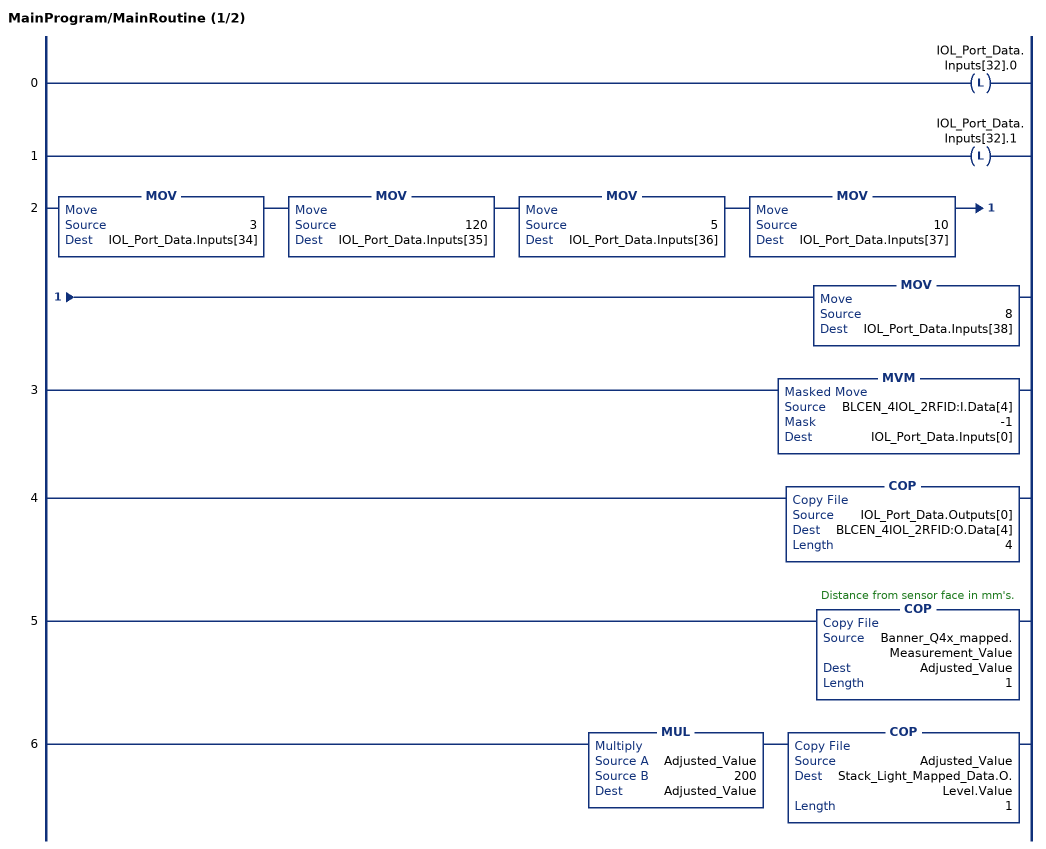
   0: OTL(IOL_Port_Data.Inputs[32].0);
   1: OTL(IOL_Port_Data.Inputs[32].1);
   2: MOV(3,IOL_Port_Data.Inputs[34])MOV(120,IOL_Port_Data.Inputs[35])MOV(5,IOL_Port_Data.Inputs[36])MOV(10,IOL_Port_Data.Inputs[37])MOV(8,IOL_Port_Data.Inputs[38]);
   3: MVM(BLCEN_4IOL_2RFID:I.Data[4],-1,IOL_Port_Data.Inputs[0]);
   4: COP(IOL_Port_Data.Outputs[0],BLCEN_4IOL_2RFID:O.Data[4],4);
   5: COP(Banner_Q4x_mapped.Measurement_Value,Adjusted_Value,1);
   6: MUL(Adjusted_Value,200,Adjusted_Value)COP(Adjusted_Value,Stack_Light_Mapped_Data.O.Level.Value,1);
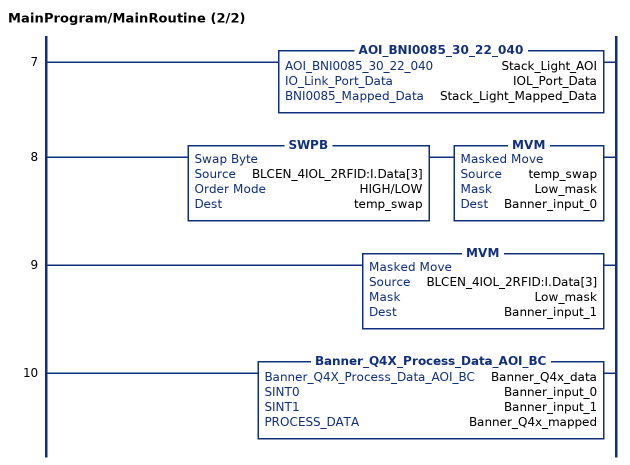
   7: AOI_BNI0085_30_22_040(Stack_Light_AOI,IOL_Port_Data,Stack_Light_Mapped_Data);
   8: SWPB(BLCEN_4IOL_2RFID:I.Data[3],HIGH/LOW,temp_swap)MVM(temp_swap,Low_mask,Banner_input_0);
   9: MVM(BLCEN_4IOL_2RFID:I.Data[3],Low_mask,Banner_input_1);
   10: Banner_Q4X_Process_Data_AOI_BC(Banner_Q4x_data,Banner_input_0,Banner_input_1,Banner_Q4x_mapped);
END_ROUTINE
END_PROGRAM

PROGRAM SafetyProgram   (* main routine MainRoutine, safety *)

ROUTINE MainRoutine   (* ladder *)
END_ROUTINE
END_PROGRAM
